% RSLogix 500 project PROJECT8_PID_SUBSTITUTION.RSS, saved by version 8.30.00.16 %
PROJECT "UNTITLED"    % processor: Bul.1763 MicroLogix 1100 Series B %

PROGRAM FILES
  LAD 2 "MAIN"  2 rungs
  LAD 3 "CONTROL"  18 rungs

DATA FILES
  O0 OUTPUT  4 elements
  I1 INPUT  6 elements
  S2 STATUS  66 elements
  B3 BINARY  1 elements
  T4 TIMER  1 elements
  C5 COUNTER  1 elements
  R6 CONTROL  1 elements
  N7 INTEGER  7 elements
  F8 FLOAT  1 elements

LADDER 2 "MAIN"
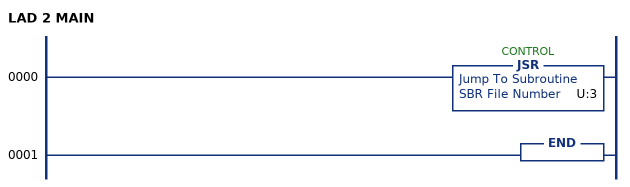
% Rung: 0 %
SOR JSR U:3 EOR
%   U:3  "CONTROL" %
% Rung: 1 %
SOR END EOR

LADDER 3 "CONTROL"
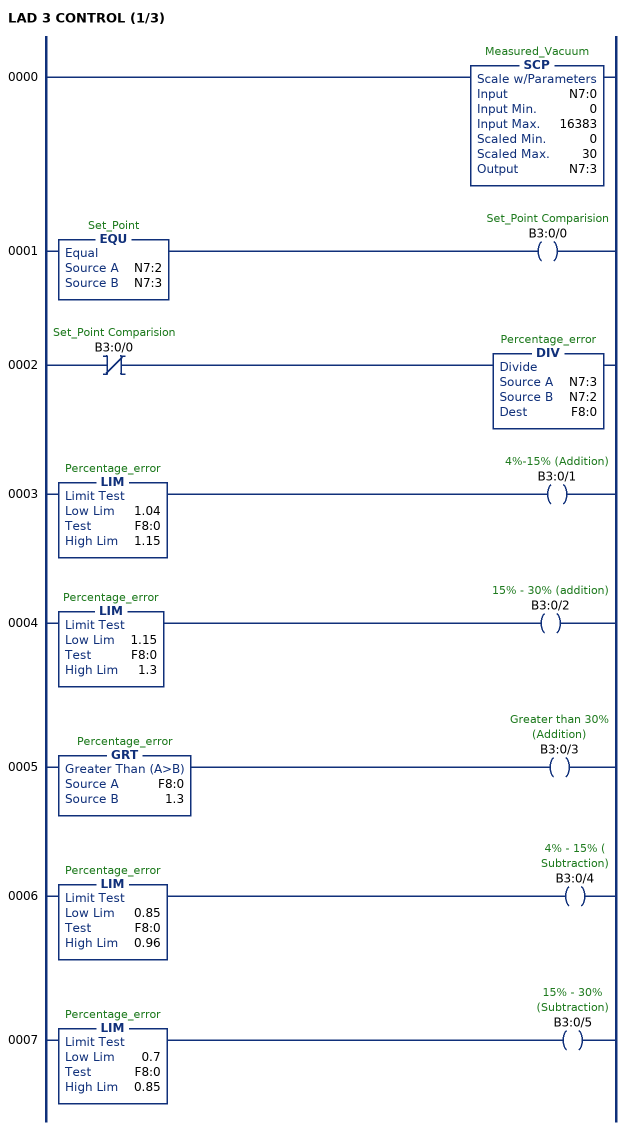
% Rung: 0 %
SOR SCP N7:0 0 16383 0 30 N7:3 EOR
%   N7:0  "input" %
%   N7:3  "Measured_Vacuum" %
% Rung: 1 %
SOR EQU N7:2 N7:3 OTE B3:0/0 EOR
%   N7:2  "Set_Point" %
%   N7:3  "Measured_Vacuum" %
%   B3:0/0  "Set_Point Comparision" %
% Rung: 2 %
SOR XIO B3:0/0 DIV N7:3 N7:2 F8:0 EOR
%   B3:0/0  "Set_Point Comparision" %
%   N7:3  "Measured_Vacuum" %
%   N7:2  "Set_Point" %
%   F8:0  "Percentage_error" %
% Rung: 3 %
SOR LIM 1.04 F8:0 1.15 OTE B3:0/1 EOR
%   F8:0  "Percentage_error" %
%   B3:0/1  "4%-15% (Addition)" %
% Rung: 4 %
SOR LIM 1.15 F8:0 1.3 OTE B3:0/2 EOR
%   F8:0  "Percentage_error" %
%   B3:0/2  "15% - 30% (addition)" %
% Rung: 5 %
SOR GRT F8:0 1.3 OTE B3:0/3 EOR
%   F8:0  "Percentage_error" %
%   B3:0/3  "Greater than 30% (Addition)" %
% Rung: 6 %
SOR LIM 0.85 F8:0 0.96 OTE B3:0/4 EOR
%   F8:0  "Percentage_error" %
%   B3:0/4  "4% - 15% (Subtraction)" %
% Rung: 7 %
SOR LIM 0.7 F8:0 0.85 OTE B3:0/5 EOR
%   F8:0  "Percentage_error" %
%   B3:0/5  "15% - 30% (Subtraction)" %

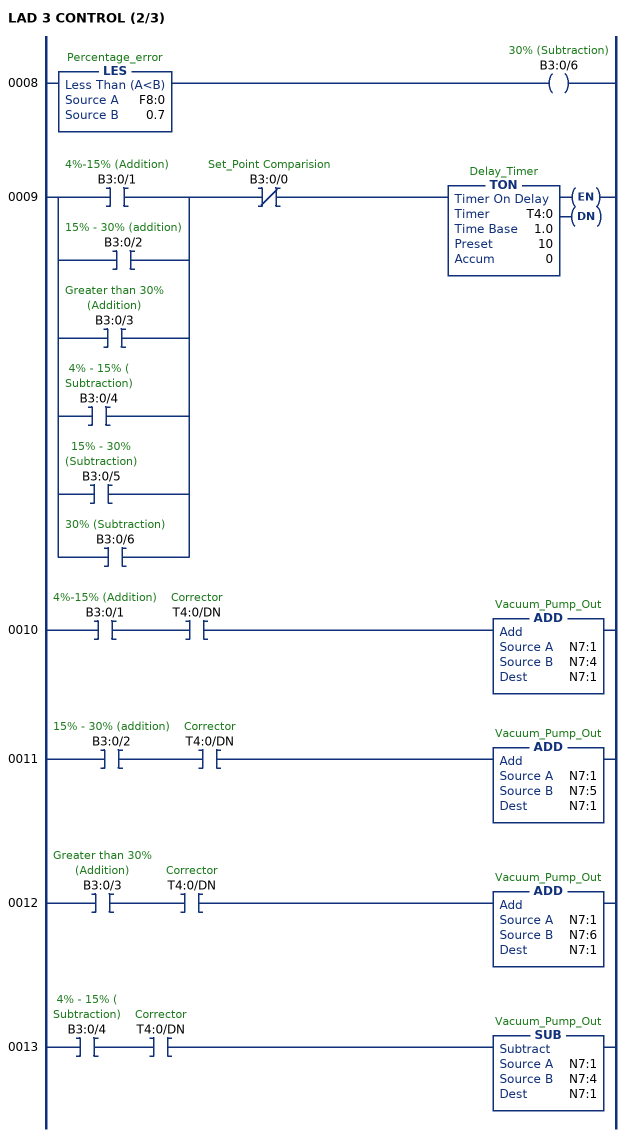
% Rung: 8 %
SOR LES F8:0 0.7 OTE B3:0/6 EOR
%   F8:0  "Percentage_error" %
%   B3:0/6  "30% (Subtraction)" %
% Rung: 9 %
SOR BST XIC B3:0/1 NXB XIC B3:0/2 NXB XIC B3:0/3 NXB XIC B3:0/4 NXB XIC B3:0/5 NXB XIC B3:0/6 BND XIO B3:0/0 TON T4:0 1.0 10 0 EOR
%   B3:0/1  "4%-15% (Addition)" %
%   B3:0/2  "15% - 30% (addition)" %
%   B3:0/3  "Greater than 30% (Addition)" %
%   B3:0/4  "4% - 15% (Subtraction)" %
%   B3:0/5  "15% - 30% (Subtraction)" %
%   B3:0/6  "30% (Subtraction)" %
%   B3:0/0  "Set_Point Comparision" %
%   T4:0  "Delay_Timer" %
% Rung: 10 %
SOR XIC B3:0/1 XIC T4:0/DN ADD N7:1 N7:4 N7:1 EOR
%   B3:0/1  "4%-15% (Addition)" %
%   T4:0/DN  "Corrector" %
%   N7:1  "Vacuum_Pump_Out" %
%   N7:4  "feedback_amend" %
% Rung: 11 %
SOR XIC B3:0/2 XIC T4:0/DN ADD N7:1 N7:5 N7:1 EOR
%   B3:0/2  "15% - 30% (addition)" %
%   T4:0/DN  "Corrector" %
%   N7:1  "Vacuum_Pump_Out" %
%   N7:5  "Value_60" %
% Rung: 12 %
SOR XIC B3:0/3 XIC T4:0/DN ADD N7:1 N7:6 N7:1 EOR
%   B3:0/3  "Greater than 30% (Addition)" %
%   T4:0/DN  "Corrector" %
%   N7:1  "Vacuum_Pump_Out" %
%   N7:6  "Value_100" %
% Rung: 13 %
SOR XIC B3:0/4 XIC T4:0/DN SUB N7:1 N7:4 N7:1 EOR
%   B3:0/4  "4% - 15% (Subtraction)" %
%   T4:0/DN  "Corrector" %
%   N7:1  "Vacuum_Pump_Out" %
%   N7:4  "feedback_amend" %

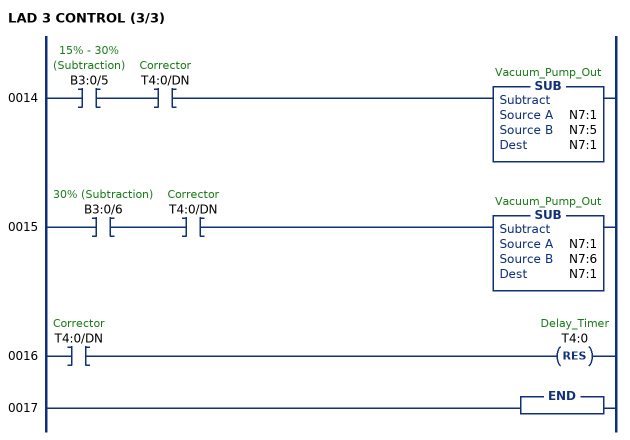
% Rung: 14 %
SOR XIC B3:0/5 XIC T4:0/DN SUB N7:1 N7:5 N7:1 EOR
%   B3:0/5  "15% - 30% (Subtraction)" %
%   T4:0/DN  "Corrector" %
%   N7:1  "Vacuum_Pump_Out" %
%   N7:5  "Value_60" %
% Rung: 15 %
SOR XIC B3:0/6 XIC T4:0/DN SUB N7:1 N7:6 N7:1 EOR
%   B3:0/6  "30% (Subtraction)" %
%   T4:0/DN  "Corrector" %
%   N7:1  "Vacuum_Pump_Out" %
%   N7:6  "Value_100" %
% Rung: 16 %
SOR XIC T4:0/DN RES T4:0 EOR
%   T4:0/DN  "Corrector" %
%   T4:0  "Delay_Timer" %
% Rung: 17 %
SOR END EOR

DATA TABLE (non-zero values as saved)
DATA T4
% .PRE .ACC %
% T4:0 % 10 0
